VAR_GLOBAL
END_VAR

(* stored: Version 1.1.0.1, ProductVersion 3.1.0.19
   GVL CHD_CmdState: Id {1054af7f-24de-44c2-bb11-e55bbf723053} *)
